SUBAPPLICATION Uebung_019b (* Umschalten einer Maske *)
  (* Standard: 61499-2; Description: Copyright (c) 2023 Meisterschulen am Ostbahnhof This program and the accompanying materials are made available under the terms of the Eclipse Public License 2.0 which is available at https://www.eclipse.org/legal/epl-2.0/ SPDX-License-Identifier: EPL-2.0 *)
  (* Version 1.0, 2023-10-23, Franz Höpfinger, Meisterschulen am Ostbahnhof *)
  IMPORT logiBUS::io::DI::logiBUS_DI;
  IMPORT logiBUS::io::DQ::logiBUS_DO;
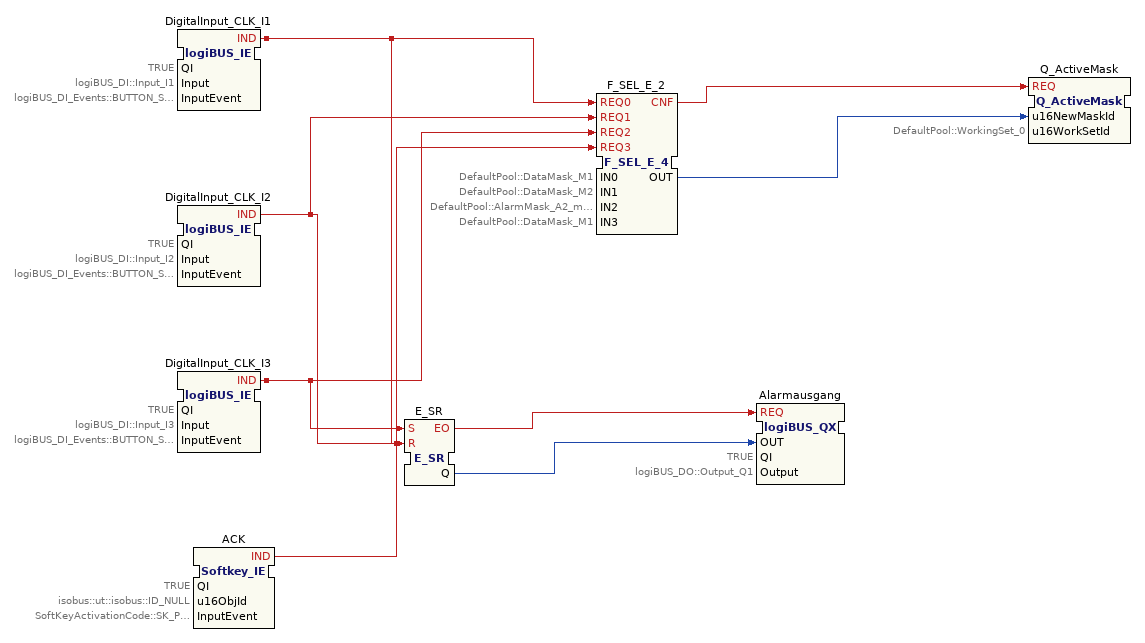
  FBS
    DigitalInput_CLK_I1 : logiBUS_IE(QI := TRUE, Input := logiBUS_DI::Input_I1, InputEvent := logiBUS_DI_Events::BUTTON_SINGLE_CLICK);
    Q_ActiveMask : isobus::ut::Q_ActiveMask(u16WorkSetId := DefaultPool::WorkingSet_0);
    DigitalInput_CLK_I2 : logiBUS_IE(QI := TRUE, Input := logiBUS_DI::Input_I2, InputEvent := logiBUS_DI_Events::BUTTON_SINGLE_CLICK);
    F_SEL_E_2 : F_SEL_E_4(IN0 := DefaultPool::DataMask_M1, IN1 := DefaultPool::DataMask_M2, IN2 := DefaultPool::AlarmMask_A2_medium, IN3 := DefaultPool::DataMask_M1);
    DigitalInput_CLK_I3 : logiBUS_IE(QI := TRUE, Input := logiBUS_DI::Input_I3, InputEvent := logiBUS_DI_Events::BUTTON_SINGLE_CLICK);
    ACK : Softkey_IE(QI := TRUE, u16ObjId := isobus::ut::isobus::ID_NULL, InputEvent := SoftKeyActivationCode::SK_PRESSED);
    E_SR : iec61499::events::E_SR;
    Alarmausgang : logiBUS::io::DQ::logiBUS_QX(QI := TRUE, Output := logiBUS_DO::Output_Q1);
  END_FBS
  EVENT_CONNECTIONS
    DigitalInput_CLK_I1.IND TO F_SEL_E_2.REQ0;
    DigitalInput_CLK_I2.IND TO F_SEL_E_2.REQ1;
    F_SEL_E_2.CNF TO Q_ActiveMask.REQ;
    DigitalInput_CLK_I3.IND TO F_SEL_E_2.REQ2;
    ACK.IND TO F_SEL_E_2.REQ3;
    DigitalInput_CLK_I3.IND TO E_SR.S;
    DigitalInput_CLK_I2.IND TO E_SR.R;
    DigitalInput_CLK_I1.IND TO E_SR.R;
    ACK.IND TO E_SR.R;
    E_SR.EO TO Alarmausgang.REQ;
  END_CONNECTIONS
  DATA_CONNECTIONS
    F_SEL_E_2.OUT TO Q_ActiveMask.u16NewMaskId;
    E_SR.Q TO Alarmausgang.OUT;
  END_CONNECTIONS
END_SUBAPPLICATION
